FUNCTION_BLOCK TcoRtcTest EXTENDS TcoCore._internals_TcoContext
VAR
    _callMyPlcInstanceSync : BOOL := FALSE;
    _callMyPlcInstanceRun : BOOL := FALSE;
    _myIdentity : ULINT;
    _nowLocal : DATE_AND_TIME;
    _nowUtc : DATE_AND_TIME;
    _rtcIsValid : BOOL := FALSE;
    _rtcIsSynchronized : BOOL := FALSE;
    _rtcSynchParamsSet : TcoCore.RtcSynchParams;
    _rtcSynchParamsGet : TcoCore.RtcSynchParams;
END_VAR

IF THIS^._callMyPlcInstanceSync THEN
    THIS^.RtcSynchronize(_rtcSynchParamsSet.doSynch, _rtcSynchParamsSet.syncAmsId, _rtcSynchParamsSet.syncPeriod);
END_IF

IF THIS^._callMyPlcInstanceRun THEN
    THIS^.Run();
    _nowLocal := THIS^.RealTimeClock.NowLocal();
    _nowUtc := THIS^.RealTimeClock.NowUTC();
    _rtcIsValid := THIS^.RealTimeClock.IsValid;
    _rtcIsSynchronized := THIS^.RealTimeClock.IsSynchronized;
    _myIdentity := THIS^.Identity;
END_IF

{attribute 'TcRpcEnable'}
METHOD INTERNAL GetSynchParams
_rtcSynchParamsGet := SUPER^._GetSynchParams();
END_METHOD

METHOD PROTECTED Main
END_METHOD

{attribute 'TcRpcEnable'}
METHOD INTERNAL NowLocal
_nowLocal := THIS^.RealTimeClock.NowLocal();
END_METHOD

{attribute 'TcRpcEnable'}
METHOD INTERNAL NowUtc
_nowUtc := THIS^.RealTimeClock.NowUTC();
END_METHOD

{attribute 'TcRpcEnable'}
METHOD INTERNAL RtcIsSynchronized : BOOL
RtcIsSynchronized := THIS^.RealTimeClock.IsSynchronized;
_rtcIsSynchronized := THIS^.RealTimeClock.IsSynchronized;
END_METHOD

{attribute 'TcRpcEnable'}
METHOD INTERNAL RtcIsValid : BOOL
RtcIsValid := THIS^.RealTimeClock.IsValid;
_rtcIsValid := THIS^.RealTimeClock.IsValid;
END_METHOD

{attribute 'TcRpcEnable'}
METHOD INTERNAL TickClock : STRING
TickClock := Tc2_EtherCAT.DCTIME64_TO_STRING(THIS^.RealTimeClock.TickClock());
END_METHOD

END_FUNCTION_BLOCK

(* stored: Version 1.1.0.1
   POU TcoRtcTest: Id {422101bf-9bdb-02c4-0505-5d211f35b9e7}, SpecialFunc None
   Method GetSynchParams: Id {43774be5-16e1-0926-1900-f0d18d06faf5}
   Method Main: Id {ab154a48-9ac1-0c37-230b-2e533fa7520e}
   Method NowLocal: Id {f0f7feae-fd4c-0752-2e52-d4f3673f6f89}
   Method NowUtc: Id {4d15ee95-7f3e-081c-2de7-138c5254d6a7}
   Method RtcIsSynchronized: Id {9de41ec0-7d16-00fc-36c5-1766b55aec78}
   Method RtcIsValid: Id {afc935ba-1696-0021-0046-4e4809990779}
   Method TickClock: Id {396b1245-0012-0d3d-2e99-6b4b82f03984} *)
